RoboDK station: Nemo_tool_test(1).rdk

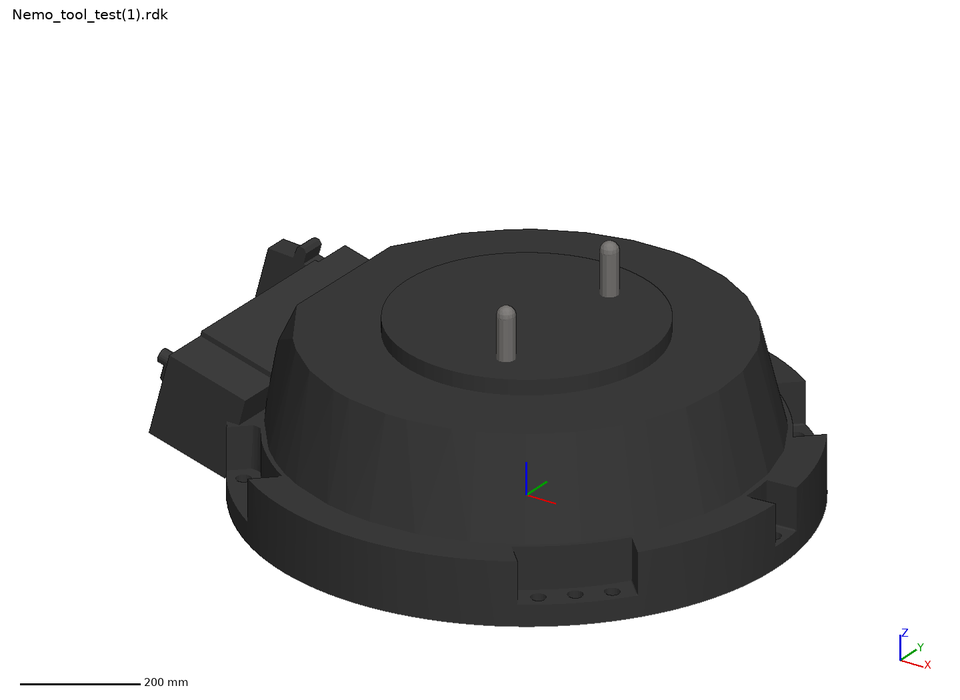
[picture v0: the station drawn from its stored meshes, robots at their saved joint values, targets as dots, program paths as lines]
Station Nemo_tool_test (saved by RoboDK 5.4.2). Poses are relative to the parent item; angles as X-Y-Z fixed-axis rotations.
  - frame KUKA KR 210-2 Base at (0, 0, 0) mm
    - robot KUKA KR 210-2: 6 axes, payload 210 kg, reach 2700 mm, repeatability 0.06 mm, weight 1267 kg
        joint limits [-185, -146, -119, -350, -125, -350] to [185, 0, 155, 350, 125, 350]; home [0, -90, 90, 0, 0, 0]; saved at [0, -82.167, 106.498, 0, -24.332, 0]
      - tool NEMO_TOOL, TCP at (0, 0, 0) mm, size 350 x 500 x 427.5 mm, geometry from NEMO_TOOL.step
